// TwinCAT 3 PLC project Cordinator
// ProgramVersion: 3.1.4026.23
// libraries:
//   Tc2_Standard, * (Beckhoff Automation GmbH)
//   Tc2_System, * (Beckhoff Automation GmbH)
//   Tc2_Utilities, * (Beckhoff Automation GmbH)
// project tree:
//   / cppTask.TcTTO, PlcTask.TcTTO
//   POUs/ F_WriteDataArea.TcPOU, PRG_Cpp_Cordinator.TcPOU, PRG_PLC_Cordinator.TcPOU, TComGetModulesByClass.TcPOU
// (motion and I/O tree: see PLC project plc)
// real-time tasks:
//   TASK PlcTask: cycle T#10ms, priority 20, ADS port 350
//   TASK cppTask: cycle T#10ms, priority 15, ADS port 351
// variable links:

CONFIGURATION Cordinator
    RESOURCE PLC ON TwinCAT3
        TASK cppTask(INTERVAL := T#10ms, PRIORITY := 15);
        TASK PlcTask(INTERVAL := T#10ms, PRIORITY := 20);
        PROGRAM PRG_Cpp_Cordinator WITH cppTask : PRG_Cpp_Cordinator;
        PROGRAM PRG_PLC_Cordinator WITH PlcTask : PRG_PLC_Cordinator;
    END_RESOURCE
END_CONFIGURATION

// ---- POUs/PRG_Cpp_Cordinator.TcPOU
PROGRAM PRG_Cpp_Cordinator
VAR
	execute			: BOOL := FALSE;
	Step			: UDINT;
	GetPlCInstances : TComGetModulesByClass; //Ask the object server for a list of object ID's based on the class ID.
	ObjIds			: ARRAY[0..2] OF OTCID;	 // All cpp instances Object ID's - including this instnace
	NewCounterValue : UDINT;
	i				: UDINT;
END_VAR

VAR CONSTANT
	cpp_CLASS_ID : CLSID := STRING_TO_GUID('B7173B55-43BF-B00D-AA6B-FF13D43F5ECC');
	DATA_AREA_NUM : UDINT := 1;
	OFFSET		  : UDINT := 0;	
END_VAR

//Automatic on system start - after a delay
CASE Step OF
	0: //Wait for the system to startup
		IF execute THEN
			execute := FALSE;
			Step	:= 10;
		END_IF

	10: //Ask for a list of PLC object ID's
		GetPlCInstances(Execute := TRUE, ClassID := cpp_CLASS_ID, ObjectIDs := ObjIds);
		IF NOT GetPlCInstances.Busy THEN
			IF NOT GetPlCInstances.Error THEN
				Step := 20;
			END_IF

			GetPlCInstances(Execute := FALSE, ClassID := cpp_CLASS_ID, ObjectIDs := ObjIds);
		END_IF

	20: //Check if we got Object ID's of all obecjts
		Step := 30;
		FOR i := 0 TO 2 DO
			IF ObjIds[i] = 0 THEN
				Step := 10; // Try again
			END_IF
		END_FOR

	30: //Write the counters of to 0
		FOR i := 0 TO 2 DO
			F_WriteDataArea(ObjectID := ObjIds[i],
							AreaNum	 := DATA_AREA_NUM,
							OffSet	 := OFFSET,
							Size	 := SIZEOF(NewCounterValue),
							pData	 := ADR(NewCounterValue));
		END_FOR

		Step := 40;

	40:
		;
END_CASE

END_PROGRAM

// ---- POUs/TComGetModulesByClass.TcPOU
{attribute 'hide_all_locals'}
FUNCTION_BLOCK TComGetModulesByClass
VAR_INPUT
    Execute : BOOL;
    ClassID : CLSID;
    Library : STRING := ''; // [OPTIONAL] e.g. C++ Module Vendor|MyModule|0.0.0.1
END_VAR

VAR_IN_OUT
    ObjectIDs : ARRAY [*] OF OTCID;
END_VAR

VAR_OUTPUT
    Busy    : BOOL;
    Error   : BOOL;
    ErrorID : UDINT;
    Count   : UDINT;
END_VAR

VAR
    _onExecute          : R_TRIG;
    _getModuleObjectIDs : ADSRDWRT;

    _lowerBound : DINT;
    _upperBound : DINT;
    _dataSize   : UDINT;
    i           : DINT;
    _state      : (
        IDLE,
        EXEC,
        DONE,
        ERR
    );
    _classIdVersioned : CLSID;
END_VAR

VAR CONSTANT
    EMPTY_CLASS_ID : CLSID := STRING_TO_GUID( '00000000-0000-0000-0000-000000000000' );
	TCOM_OBJECT_SERVER_ADS_PORT : T_AmsPort := 10;
	GET_MODULES_INDEX_GROUP : UDINT := 16#201;
	GET_MODULES_INDEX_OfFSET : UDINT := 16#02;
END_VAR

_onExecute( CLK := Execute );

IF _onExecute.Q AND NOT Busy THEN
    Error   := FALSE;
    ErrorID := 0;
    Count   := 0;

    IF GuidsEqual( ADR( ClassID ), ADR( EMPTY_CLASS_ID ) ) THEN
        Error   := TRUE;
        ErrorID := E_AdsErr.DEVICE_INVALIDCLSID;
        RETURN;
    END_IF

    IF ObjectIDs = 0 THEN
        Error   := TRUE;
        ErrorID := E_AdsErr.DEVICE_INVALIDDATA;
        RETURN;
    END_IF

    _lowerBound := LOWER_BOUND( ObjectIDs, 1 );
    _upperBound := UPPER_BOUND( ObjectIDs, 1 );

    IF _lowerBound < 0 OR _upperBound < 0 THEN
        Error   := TRUE;
        ErrorID := E_AdsErr.DEVICE_INVALIDDATA;
        RETURN;
    END_IF

	_dataSize := TO_UDINT( _upperBound - _lowerBound + 1 );

    IF Library <> '' THEN
		
		IF FIND(Library, '|') = 0 THEN // invalid library format
			Error   := TRUE;
            ErrorID := E_AdsErr.DEVICE_INVALIDCLSID;
            RETURN;
		END_IF
	
        IF NOT F_GetClassIdVersioned( Library, ClassID, _classIdVersioned ) THEN
            Error   := TRUE;
            ErrorID := E_AdsErr.DEVICE_INVALIDCLSID;
            RETURN;
        END_IF
	ELSE
		_classIdVersioned := ClassID;
    END_IF

    Busy   := TRUE;
    _state := EXEC;

END_IF

CASE _state OF

    IDLE:
		Busy := FALSE;
		
		IF NOT Execute THEN
			Error := FALSE;
			ErrorID := 0;
			Count := 0;
		END_IF

    EXEC:

        _getModuleObjectIDs(
            NetID    := '',
            Port     := TCOM_OBJECT_SERVER_ADS_PORT,
            WRTRD    := TRUE,
            IDXGRP   := GET_MODULES_INDEX_GROUP,
            IDXOFFS  := GET_MODULES_INDEX_OfFSET,
            WRITELEN := SIZEOF( _classIdVersioned ),
            SRCADDR  := ADR( _classIdVersioned ),
            READLEN  := (_dataSize * SIZEOF( OTCID )),
            DESTADDR := ObjectIDs
        );

        IF NOT _getModuleObjectIDs.BUSY THEN
            IF NOT _getModuleObjectIDs.ERR THEN

                FOR i := _lowerBound TO _upperBound DO
                    IF ObjectIDs[i] <> 0 THEN
                        Count := Count + 1;
                    END_IF
                END_FOR

                _state := DONE;
            ELSE
                ErrorID := _getModuleObjectIDs.ERRID;
                _state  := ERR;
            END_IF

            _getModuleObjectIDs( WRTRD := FALSE );
        END_IF

    DONE:
        Busy   := FALSE;
        _state := IDLE;

    ERR:
        Error  := TRUE;
        Busy   := FALSE;
        _state := IDLE;

END_CASE

END_FUNCTION_BLOCK

// ---- POUs/F_WriteDataArea.TcPOU
FUNCTION F_WriteDataArea : HRESULT
VAR_INPUT
	ObjectID : OTCID;
	AreaNum	 : UDINT;
	OffSet	 : UDINT;
	Size	 : UDINT;
	pData	 : PVOID;
END_VAR

VAR
	_ipDataArea : ITCADI;
	_hr			: HRESULT;
	_pData		: POINTER TO PVOID;
END_VAR

VAR CONSTANT
	IID_ITcADI : IID := TC_GLOBAL_IID_LIST.IID_ITcADI;
END_VAR

_hr := S_OK;
IF ObjectID = 0 THEN
	_hr				:= E_AdsErr.DEVICE_INVALIDDATA;
	F_WriteDataArea := _hr;
	RETURN;
END_IF

_hr := FW_ObjMgr_GetObjectInstance(oid := ObjectID, iid := IID_ITcADI, ADR(_ipDataArea));
IF _hr <> S_OK THEN
	F_WriteDataArea := _hr;
	RETURN;
END_IF

_hr := _ipDataArea.GetImagePtr(size	  := Size,
							   offs	  := OffSet,
							   adi_x  := AreaNum,
							   ppData := ADR(_pData));

IF _hr = S_OK THEN
	MEMCPY(destAddr := _pData, srcAddr := pData, n := Size);
	_hr := _ipDataArea.ReleaseImagePtr(_pData);
END_IF

_hr				:= FW_SafeRelease(ADR(_ipDataArea));
F_WriteDataArea := _hr;

END_FUNCTION

// ---- POUs/PRG_PLC_Cordinator.TcPOU
PROGRAM PRG_PLC_Cordinator
VAR
	execute			: BOOL := FALSE;
	Step			: UDINT;
	GetPlCInstances : TComGetModulesByClass; //Ask the object server for a list of object ID's based on the class ID.
	ObjIds			: ARRAY[0..3] OF OTCID;	 // All PLC instances Object ID's - including this instnace
	NewCounterValue : UDINT;
	i				: UDINT;
END_VAR

VAR CONSTANT
	PLC_CLASS_ID  : CLSID := STRING_TO_GUID('08500001-0000-0000-F000-000000000064');
	DATA_AREA_NUM : UDINT := 1;
	OFFSET		  : UDINT := 387124;
END_VAR

CASE Step OF
	0:
		IF execute THEN
			execute := FALSE;
			Step	:= 10;
		END_IF

	10: //Ask for a list of PLC object ID's
		GetPlCInstances(Execute := TRUE, ClassID := PLC_CLASS_ID, ObjectIDs := ObjIds);
		IF NOT GetPlCInstances.Busy THEN
			IF NOT GetPlCInstances.Error THEN
				Step := 20;
			END_IF

			GetPlCInstances(Execute := FALSE, ClassID := PLC_CLASS_ID, ObjectIDs := ObjIds);
		END_IF

	20: //Check if we got Object ID's of all obecjts
		Step := 30;
		FOR i := 0 TO 3 DO
			IF ObjIds[i] = 0 THEN
				Step := 10; // Try again
			END_IF
		END_FOR

	30: //Write the counters of all the PLC's to 0
		FOR i := 0 TO 3 DO
			IF ObjIds[i] <> _AppInfo.ObjId THEN
				F_WriteDataArea(ObjectID := ObjIds[i],
								AreaNum	 := DATA_AREA_NUM,
								OffSet	 := OFFSET,
								Size	 := SIZEOF(NewCounterValue),
								pData	 := ADR(NewCounterValue));
			END_IF
		END_FOR

		Step := 40;

	40:
	;
END_CASE

END_PROGRAM
